(* LS Electric XG5000 project: test cps *)
(* PLC LSPLC *)
(* module base 0 slot 0: FEnet:XGL-EFMT(B) (Fast Ethernet 통신 모듈, 전기 Master) *)
VAR_GLOBAL
    T0 : TON;
    T1 : TON;
    T2 : TON;
    T3 : TON;
    T4 : TON;
    TP0 : TP;
    TP1 : TP;
    TP2 : TP;
    TP3 : TP;
END_VAR

(* Comments on direct variables
%MW0	1 comID
%MW1	2 comID
%MW2	3 comID
%MW3	4 comID
%MW4	5 comID
%MW5	6 comID
%MW6	7 comID
%MW7	8 comID
%MW8	1 Status
%MW9	2 Status
%MW10	3 Status
%MW11	4 Status
%MW12	5 Status
%MW13	6 Status
%MW14	7 Status
%MW15	8 Status
%MW16	1 ReadData
%MW17	2 ReadData
%MW18	3 ReadData
%MW19	4 ReadData
%MW20	5 ReadData
%MW21	6 ReadData
%MW22	7 ReadData
%MW23	8 ReadData
%MW101	1번무게합
%MW102	2번무게합
%MW103	3번무게합
%MW104	4번무게합
%MW201	리셋수(트레일러)
%MW202	리셋수(트레일러)
%MW203	리셋수(트레일러)
%MW204	리셋수(트레일러)
%QX0.0.0	Belt Conveyor 0
%QX0.0.1	Belt Conveyor 1
%QX0.0.2	Belt Conveyor 2
%QX0.0.3	box
%QX0.0.4	Belt Conveyor 4
%QX0.0.5	Belt Conveyor 5
%QX0.0.6	Belt Conveyor 6
%QX0.0.7	Belt Conveyor 7
%QX0.0.8	Belt Conveyor 8
%QX0.0.9	Belt Conveyor 9
%QX0.0.10	Belt Conveyor 10
%QX0.0.11	Belt Conveyor 11
%QX0.0.12	box
%QX0.0.13	Push 01
%QX0.0.14	Push 02
%QX0.0.15	Push 03
%QX0.0.16	Push 04
%QX0.0.17	0 Exexute
%QX0.0.18	1 Exexute
%QX0.0.19	2 Exexute
%QX0.0.20	3 Exexute
%QX0.0.21	4 Exexute
%QX0.0.22	5 Exexute
%QX0.0.23	6 Exexute
%QX0.0.24	7 Exexute
%QX0.0.25	8 Exexute
%QX0.0.26	9 Exexute
%IX0.0.0	Paused
%IX0.0.1	Reset
%IX0.0.2	Running
%IX0.0.3	write00
%IX0.0.4	write01
%IX0.0.5	1 Diffuse
%IX0.0.6	2 Diffuse
%IX0.0.7	3 Diffuse
%IX0.0.8	4 Diffuse
%IX0.0.9	5 Diffuse
%IX0.0.10	6 Diffuse
%IX0.0.11	7 Diffuse
%IX0.0.12	8 Diffuse
%IX0.0.13	1 Push front_lim
%IX0.0.14	2 Push front_lim
%IX0.0.15	3 Push front_lim
%IX0.0.16	4 Push front_lim
%WW0	0 command = write
%WW1	0 WriteData
%WW2	0 Memory Index
%WW3	9 command = write
%WW4	9 WriteData
%WW5	9 Memory Index
%WW6	1 command = Read
%WW7	1 Memory Index
%WW8	2 command = Read
%WW9	2 Memory Index
%WW10	3 command = Read
%WW11	3 Memory Index
%WW12	4 command = Read
%WW13	4 Memory Index
%WW14	5 command = Read
%WW15	5 Memory Index
%WW16	6 command = Read
%WW17	6 Memory Index
%WW18	7 command = Read
%WW19	7 Memory Index
%WW20	8 command = Read
%WW21	8 Memory Index
*)

PROGRAM NewProgram (* task: 스캔 프로그램 *)
VAR
    D0 : INT;
    D10 : INT;
    D100 : INT;
    D20 : INT;
    D200 : INT;
    sensor_0ff : TON;
    sensor_1ff : TON;
END_VAR
VAR_EXTERNAL
    T0 : TON;
    T1 : TON;
    T2 : TON;
    T3 : TON;
    T4 : TON;
    TP0 : TP;
    TP1 : TP;
    TP2 : TP;
    TP3 : TP;
END_VAR
VAR
    _t1 : BOOL;
    _t2 : BOOL;
    _t3 : BOOL;
    _t4 : BOOL;
    _t5 : BOOL;
    _t6 : BOOL;
    _t7 : BOOL;
    _t8 : BOOL;
    _t9 : BOOL;
    _e10 : R_TRIG;
    _t11 : BOOL;
    _e12 : R_TRIG;
    _t13 : BOOL;
    _e14 : R_TRIG;
    _t15 : BOOL;
    _e16 : R_TRIG;
END_VAR

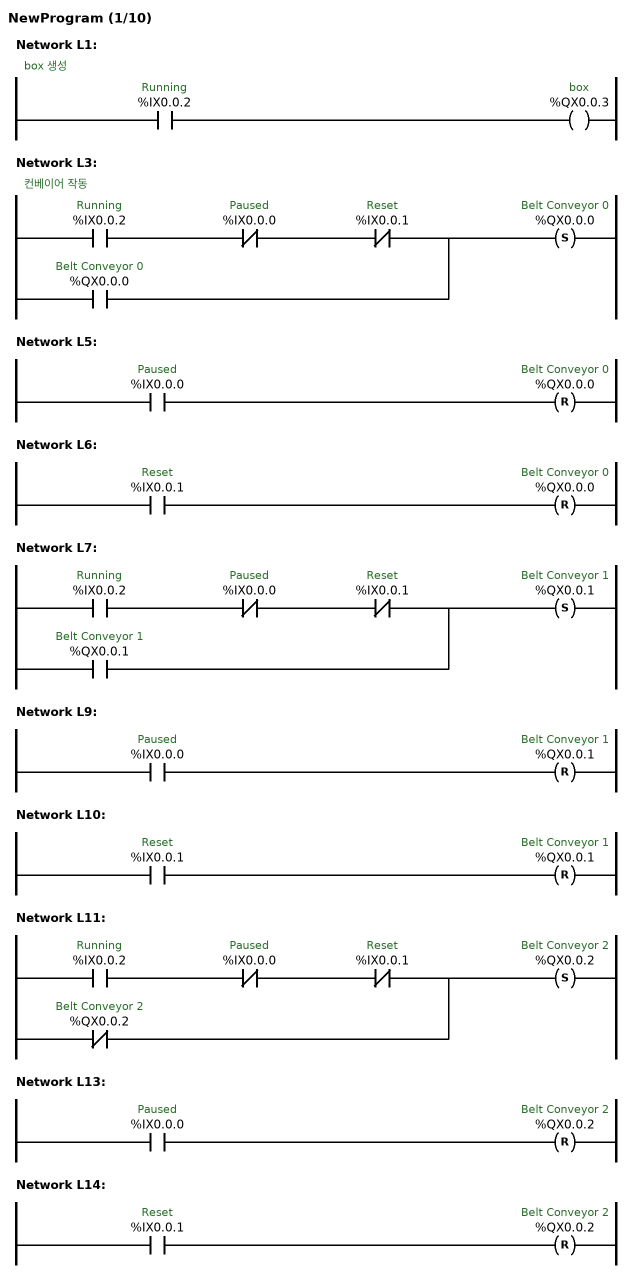
(* box 생성 *)
(* Rung L1 *)
%QX0.0.3 := %IX0.0.2;
(* 컨베이어 작동 *)
(* Rung L3 *)
IF (%IX0.0.2 AND NOT %IX0.0.0 AND NOT %IX0.0.1) OR %QX0.0.0 THEN %QX0.0.0 := TRUE; END_IF;
(* Rung L5 *)
IF %IX0.0.0 THEN %QX0.0.0 := FALSE; END_IF;
(* Rung L6 *)
IF %IX0.0.1 THEN %QX0.0.0 := FALSE; END_IF;
(* Rung L7 *)
IF (%IX0.0.2 AND NOT %IX0.0.0 AND NOT %IX0.0.1) OR %QX0.0.1 THEN %QX0.0.1 := TRUE; END_IF;
(* Rung L9 *)
IF %IX0.0.0 THEN %QX0.0.1 := FALSE; END_IF;
(* Rung L10 *)
IF %IX0.0.1 THEN %QX0.0.1 := FALSE; END_IF;
(* Rung L11 *)
IF (%IX0.0.2 AND NOT %IX0.0.0 AND NOT %IX0.0.1) OR NOT %QX0.0.2 THEN %QX0.0.2 := TRUE; END_IF;
(* Rung L13 *)
IF %IX0.0.0 THEN %QX0.0.2 := FALSE; END_IF;
(* Rung L14 *)
IF %IX0.0.1 THEN %QX0.0.2 := FALSE; END_IF;

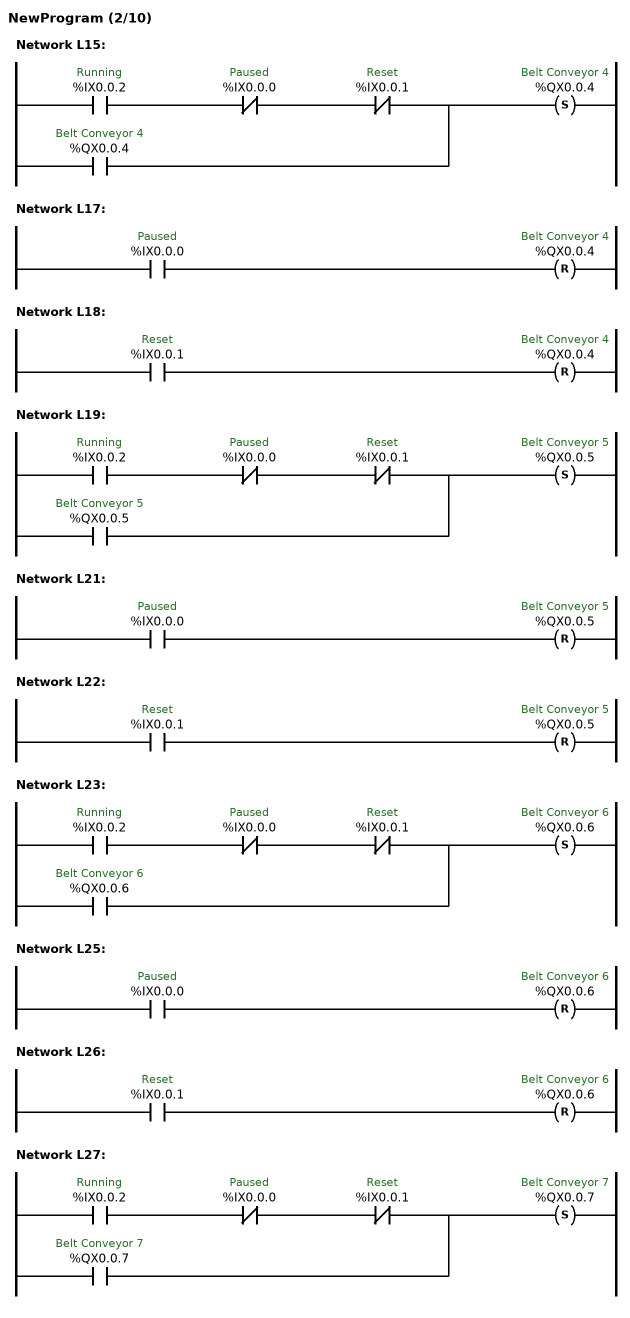
(* Rung L15 *)
IF (%IX0.0.2 AND NOT %IX0.0.0 AND NOT %IX0.0.1) OR %QX0.0.4 THEN %QX0.0.4 := TRUE; END_IF;
(* Rung L17 *)
IF %IX0.0.0 THEN %QX0.0.4 := FALSE; END_IF;
(* Rung L18 *)
IF %IX0.0.1 THEN %QX0.0.4 := FALSE; END_IF;
(* Rung L19 *)
IF (%IX0.0.2 AND NOT %IX0.0.0 AND NOT %IX0.0.1) OR %QX0.0.5 THEN %QX0.0.5 := TRUE; END_IF;
(* Rung L21 *)
IF %IX0.0.0 THEN %QX0.0.5 := FALSE; END_IF;
(* Rung L22 *)
IF %IX0.0.1 THEN %QX0.0.5 := FALSE; END_IF;
(* Rung L23 *)
IF (%IX0.0.2 AND NOT %IX0.0.0 AND NOT %IX0.0.1) OR %QX0.0.6 THEN %QX0.0.6 := TRUE; END_IF;
(* Rung L25 *)
IF %IX0.0.0 THEN %QX0.0.6 := FALSE; END_IF;
(* Rung L26 *)
IF %IX0.0.1 THEN %QX0.0.6 := FALSE; END_IF;
(* Rung L27 *)
IF (%IX0.0.2 AND NOT %IX0.0.0 AND NOT %IX0.0.1) OR %QX0.0.7 THEN %QX0.0.7 := TRUE; END_IF;

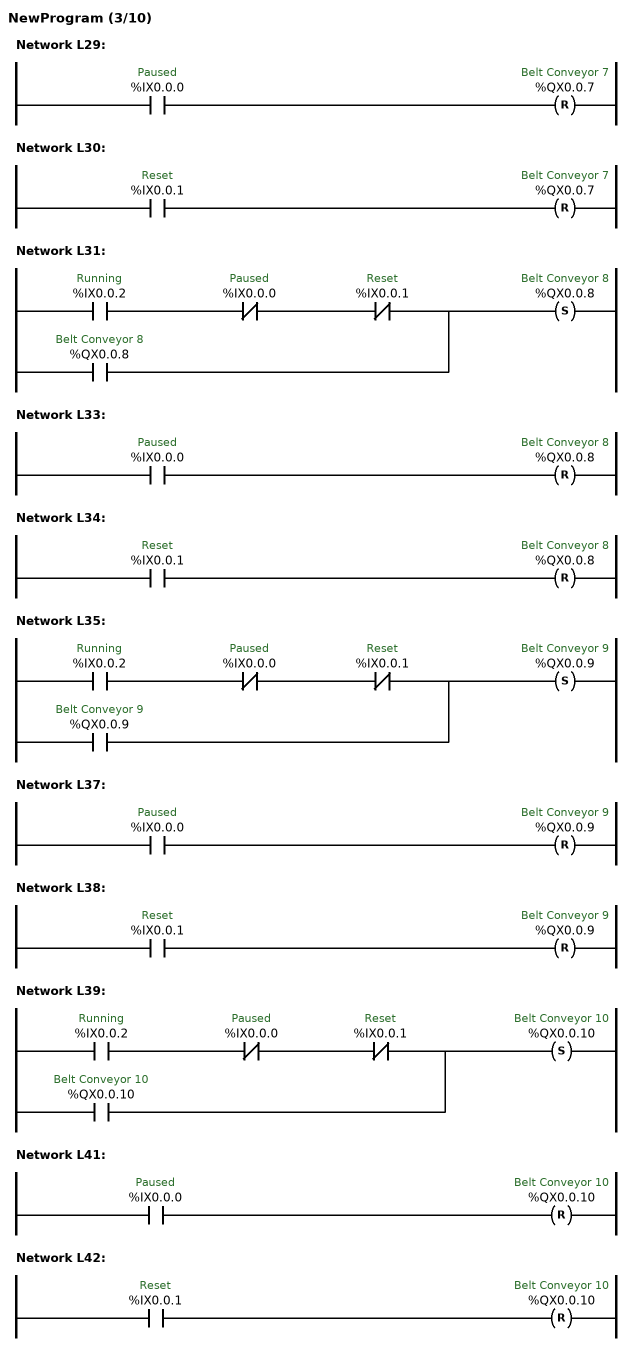
(* Rung L29 *)
IF %IX0.0.0 THEN %QX0.0.7 := FALSE; END_IF;
(* Rung L30 *)
IF %IX0.0.1 THEN %QX0.0.7 := FALSE; END_IF;
(* Rung L31 *)
IF (%IX0.0.2 AND NOT %IX0.0.0 AND NOT %IX0.0.1) OR %QX0.0.8 THEN %QX0.0.8 := TRUE; END_IF;
(* Rung L33 *)
IF %IX0.0.0 THEN %QX0.0.8 := FALSE; END_IF;
(* Rung L34 *)
IF %IX0.0.1 THEN %QX0.0.8 := FALSE; END_IF;
(* Rung L35 *)
IF (%IX0.0.2 AND NOT %IX0.0.0 AND NOT %IX0.0.1) OR %QX0.0.9 THEN %QX0.0.9 := TRUE; END_IF;
(* Rung L37 *)
IF %IX0.0.0 THEN %QX0.0.9 := FALSE; END_IF;
(* Rung L38 *)
IF %IX0.0.1 THEN %QX0.0.9 := FALSE; END_IF;
(* Rung L39 *)
IF (%IX0.0.2 AND NOT %IX0.0.0 AND NOT %IX0.0.1) OR %QX0.0.10 THEN %QX0.0.10 := TRUE; END_IF;
(* Rung L41 *)
IF %IX0.0.0 THEN %QX0.0.10 := FALSE; END_IF;
(* Rung L42 *)
IF %IX0.0.1 THEN %QX0.0.10 := FALSE; END_IF;

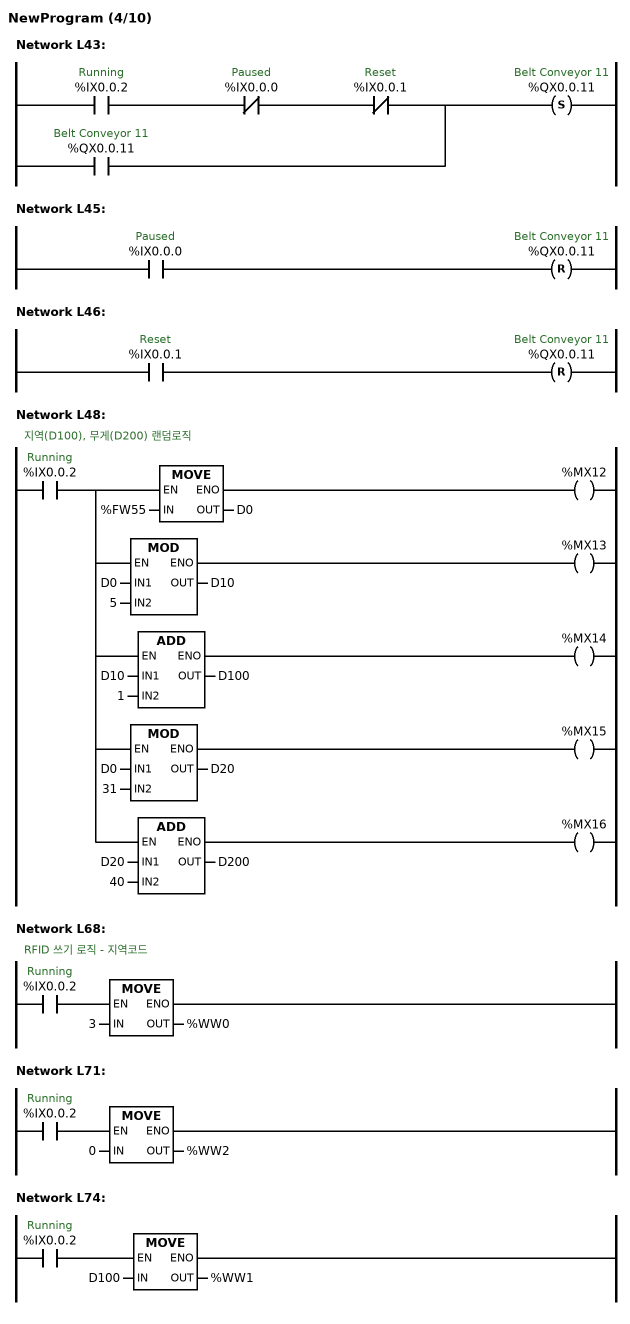
(* Rung L43 *)
IF (%IX0.0.2 AND NOT %IX0.0.0 AND NOT %IX0.0.1) OR %QX0.0.11 THEN %QX0.0.11 := TRUE; END_IF;
(* Rung L45 *)
IF %IX0.0.0 THEN %QX0.0.11 := FALSE; END_IF;
(* Rung L46 *)
IF %IX0.0.1 THEN %QX0.0.11 := FALSE; END_IF;
(* 지역(D100), 무게(D200) 랜덤로직 *)
(* Rung L48 *)
IF %IX0.0.2 THEN D0 := %FW55; END_IF;
%MX12 := %IX0.0.2;
IF %IX0.0.2 THEN D10 := D0 MOD 5; END_IF;
%MX13 := %IX0.0.2;
IF %IX0.0.2 THEN D100 := D10 + 1; END_IF;
%MX14 := %IX0.0.2;
IF %IX0.0.2 THEN D20 := D0 MOD 31; END_IF;
%MX15 := %IX0.0.2;
IF %IX0.0.2 THEN D200 := D20 + 40; END_IF;
%MX16 := %IX0.0.2;
(* RFID 쓰기 로직 - 지역코드 *)
(* Rung L68 *)
IF %IX0.0.2 THEN %WW0 := 3; END_IF;
(* Rung L71 *)
IF %IX0.0.2 THEN %WW2 := 0; END_IF;
(* Rung L74 *)
IF %IX0.0.2 THEN %WW1 := D100; END_IF;

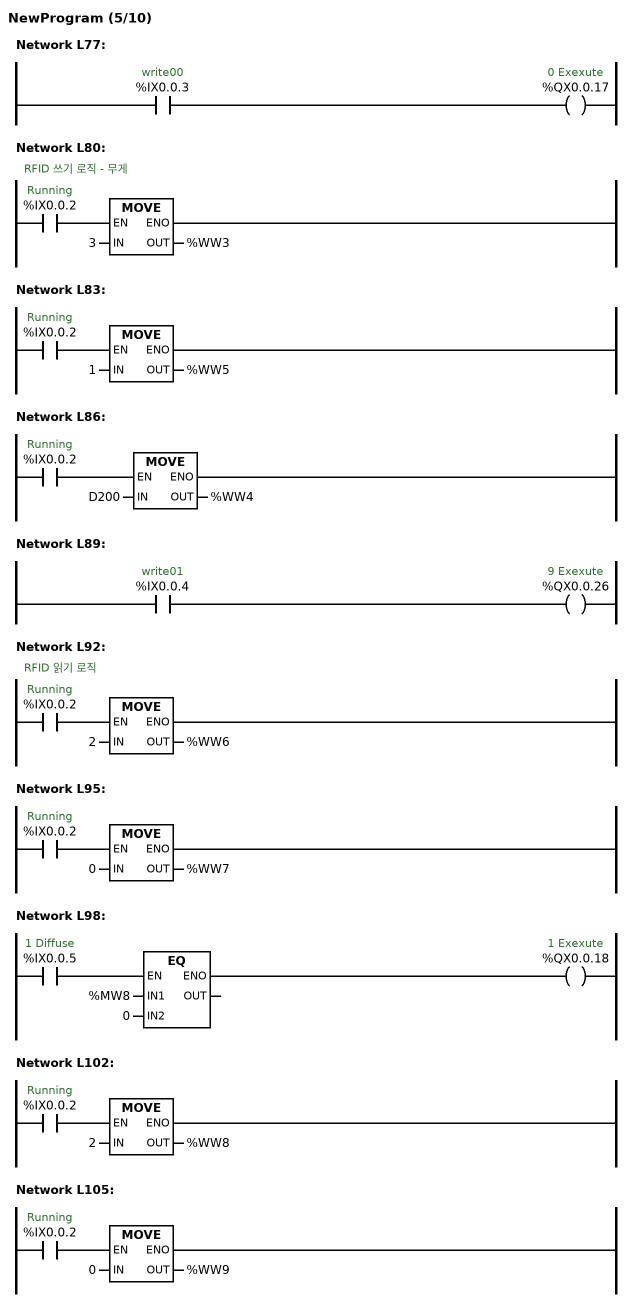
(* Rung L77 *)
%QX0.0.17 := %IX0.0.3;
(* RFID 쓰기 로직 - 무게 *)
(* Rung L80 *)
IF %IX0.0.2 THEN %WW3 := 3; END_IF;
(* Rung L83 *)
IF %IX0.0.2 THEN %WW5 := 1; END_IF;
(* Rung L86 *)
IF %IX0.0.2 THEN %WW4 := D200; END_IF;
(* Rung L89 *)
%QX0.0.26 := %IX0.0.4;
(* RFID 읽기 로직 *)
(* Rung L92 *)
IF %IX0.0.2 THEN %WW6 := 2; END_IF;
(* Rung L95 *)
IF %IX0.0.2 THEN %WW7 := 0; END_IF;
(* Rung L98 *)
IF %IX0.0.5 THEN _t1 := %MW8 = 0; END_IF;
%QX0.0.18 := %IX0.0.5;
(* Rung L102 *)
IF %IX0.0.2 THEN %WW8 := 2; END_IF;
(* Rung L105 *)
IF %IX0.0.2 THEN %WW9 := 0; END_IF;

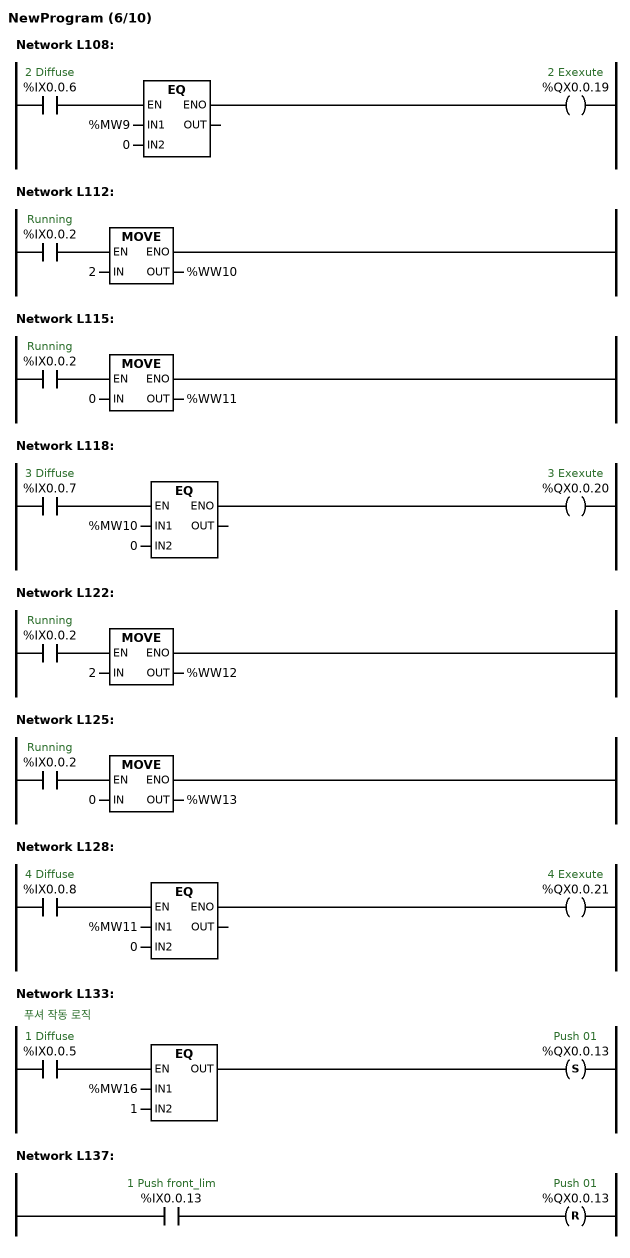
(* Rung L108 *)
IF %IX0.0.6 THEN _t2 := %MW9 = 0; END_IF;
%QX0.0.19 := %IX0.0.6;
(* Rung L112 *)
IF %IX0.0.2 THEN %WW10 := 2; END_IF;
(* Rung L115 *)
IF %IX0.0.2 THEN %WW11 := 0; END_IF;
(* Rung L118 *)
IF %IX0.0.7 THEN _t3 := %MW10 = 0; END_IF;
%QX0.0.20 := %IX0.0.7;
(* Rung L122 *)
IF %IX0.0.2 THEN %WW12 := 2; END_IF;
(* Rung L125 *)
IF %IX0.0.2 THEN %WW13 := 0; END_IF;
(* Rung L128 *)
IF %IX0.0.8 THEN _t4 := %MW11 = 0; END_IF;
%QX0.0.21 := %IX0.0.8;
(* 푸셔 작동 로직 *)
(* Rung L133 *)
IF %IX0.0.5 THEN _t5 := %MW16 = 1; END_IF;
IF _t5 THEN %QX0.0.13 := TRUE; END_IF;
(* Rung L137 *)
IF %IX0.0.13 THEN %QX0.0.13 := FALSE; END_IF;

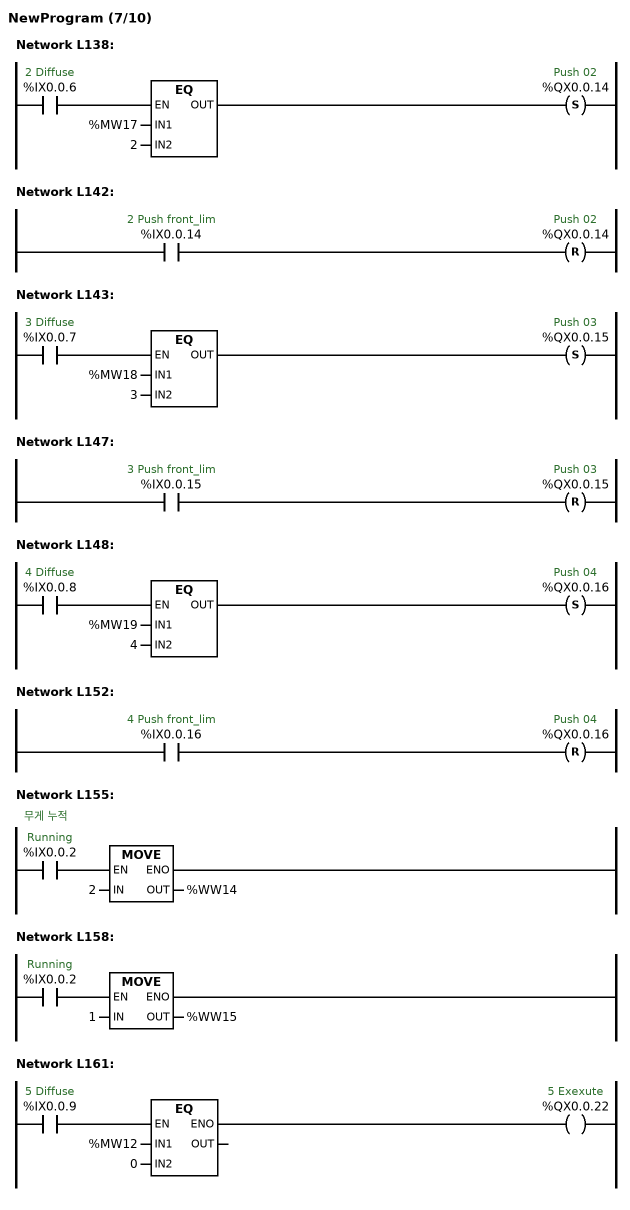
(* Rung L138 *)
IF %IX0.0.6 THEN _t6 := %MW17 = 2; END_IF;
IF _t6 THEN %QX0.0.14 := TRUE; END_IF;
(* Rung L142 *)
IF %IX0.0.14 THEN %QX0.0.14 := FALSE; END_IF;
(* Rung L143 *)
IF %IX0.0.7 THEN _t7 := %MW18 = 3; END_IF;
IF _t7 THEN %QX0.0.15 := TRUE; END_IF;
(* Rung L147 *)
IF %IX0.0.15 THEN %QX0.0.15 := FALSE; END_IF;
(* Rung L148 *)
IF %IX0.0.8 THEN _t8 := %MW19 = 4; END_IF;
IF _t8 THEN %QX0.0.16 := TRUE; END_IF;
(* Rung L152 *)
IF %IX0.0.16 THEN %QX0.0.16 := FALSE; END_IF;
(* 무게 누적 *)
(* Rung L155 *)
IF %IX0.0.2 THEN %WW14 := 2; END_IF;
(* Rung L158 *)
IF %IX0.0.2 THEN %WW15 := 1; END_IF;
(* Rung L161 *)
IF %IX0.0.9 THEN _t9 := %MW12 = 0; END_IF;
%QX0.0.22 := %IX0.0.9;

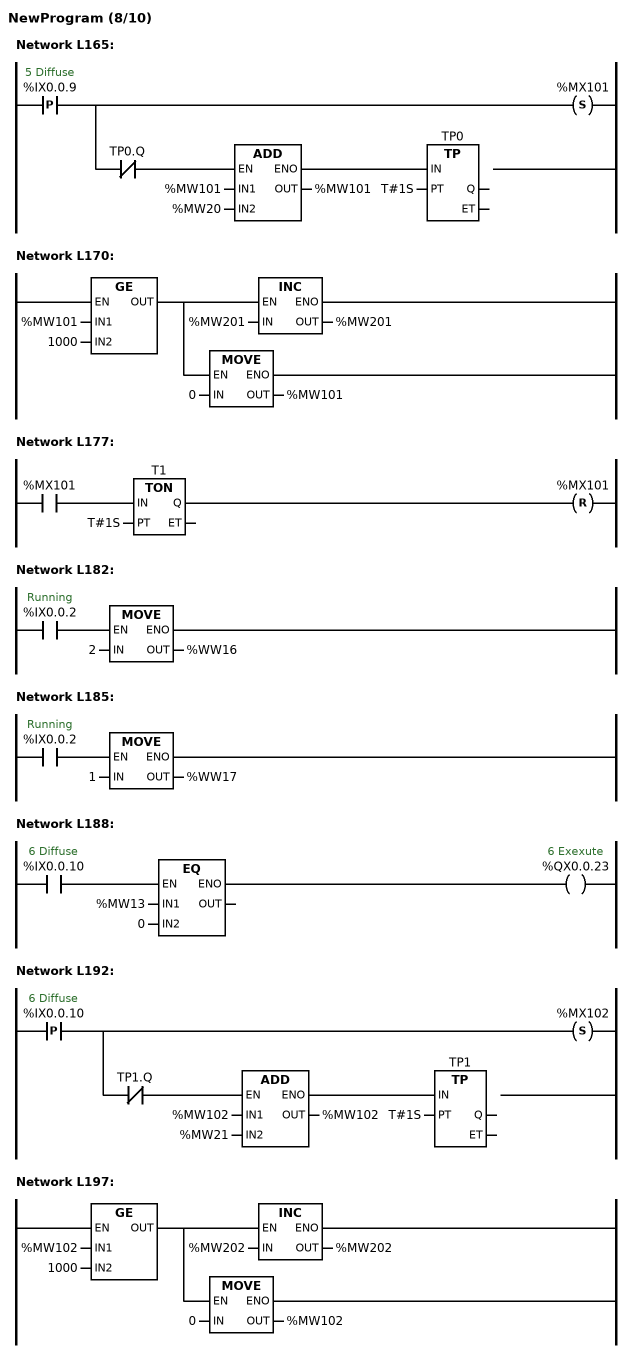
(* Rung L165 *)
_e10(CLK := %IX0.0.9);
IF _e10.Q THEN %MX101 := TRUE; END_IF;
IF _e10.Q AND NOT TP0.Q THEN %MW101 := %MW101 + %MW20; END_IF;
TP0(IN := _e10.Q AND NOT TP0.Q, PT := T#1S);
(* Rung L170 *)
IF %MW101 >= 1000 THEN
    %MW201 := INC(%MW201);
    %MW101 := 0;
END_IF;
(* Rung L177 *)
T1(IN := %MX101, PT := T#1S);
IF T1.Q THEN %MX101 := FALSE; END_IF;
(* Rung L182 *)
IF %IX0.0.2 THEN %WW16 := 2; END_IF;
(* Rung L185 *)
IF %IX0.0.2 THEN %WW17 := 1; END_IF;
(* Rung L188 *)
IF %IX0.0.10 THEN _t11 := %MW13 = 0; END_IF;
%QX0.0.23 := %IX0.0.10;
(* Rung L192 *)
_e12(CLK := %IX0.0.10);
IF _e12.Q THEN %MX102 := TRUE; END_IF;
IF _e12.Q AND NOT TP1.Q THEN %MW102 := %MW102 + %MW21; END_IF;
TP1(IN := _e12.Q AND NOT TP1.Q, PT := T#1S);
(* Rung L197 *)
IF %MW102 >= 1000 THEN
    %MW202 := INC(%MW202);
    %MW102 := 0;
END_IF;

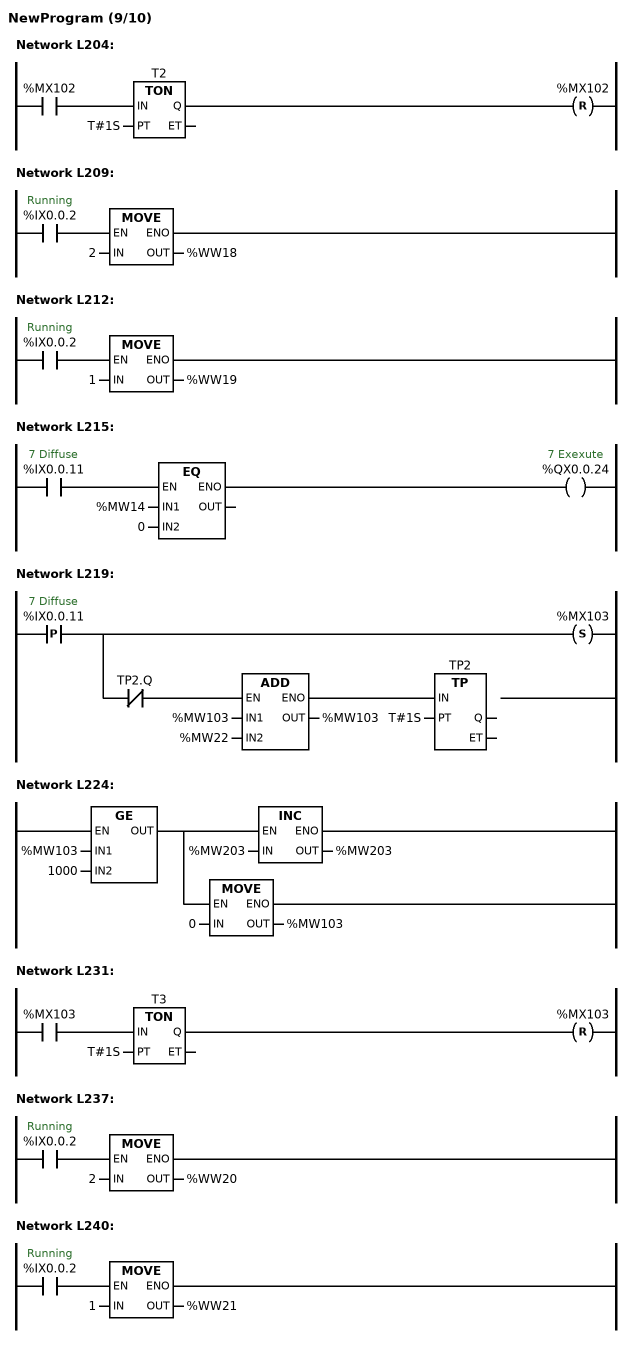
(* Rung L204 *)
T2(IN := %MX102, PT := T#1S);
IF T2.Q THEN %MX102 := FALSE; END_IF;
(* Rung L209 *)
IF %IX0.0.2 THEN %WW18 := 2; END_IF;
(* Rung L212 *)
IF %IX0.0.2 THEN %WW19 := 1; END_IF;
(* Rung L215 *)
IF %IX0.0.11 THEN _t13 := %MW14 = 0; END_IF;
%QX0.0.24 := %IX0.0.11;
(* Rung L219 *)
_e14(CLK := %IX0.0.11);
IF _e14.Q THEN %MX103 := TRUE; END_IF;
IF _e14.Q AND NOT TP2.Q THEN %MW103 := %MW103 + %MW22; END_IF;
TP2(IN := _e14.Q AND NOT TP2.Q, PT := T#1S);
(* Rung L224 *)
IF %MW103 >= 1000 THEN
    %MW203 := INC(%MW203);
    %MW103 := 0;
END_IF;
(* Rung L231 *)
T3(IN := %MX103, PT := T#1S);
IF T3.Q THEN %MX103 := FALSE; END_IF;
(* Rung L237 *)
IF %IX0.0.2 THEN %WW20 := 2; END_IF;
(* Rung L240 *)
IF %IX0.0.2 THEN %WW21 := 1; END_IF;

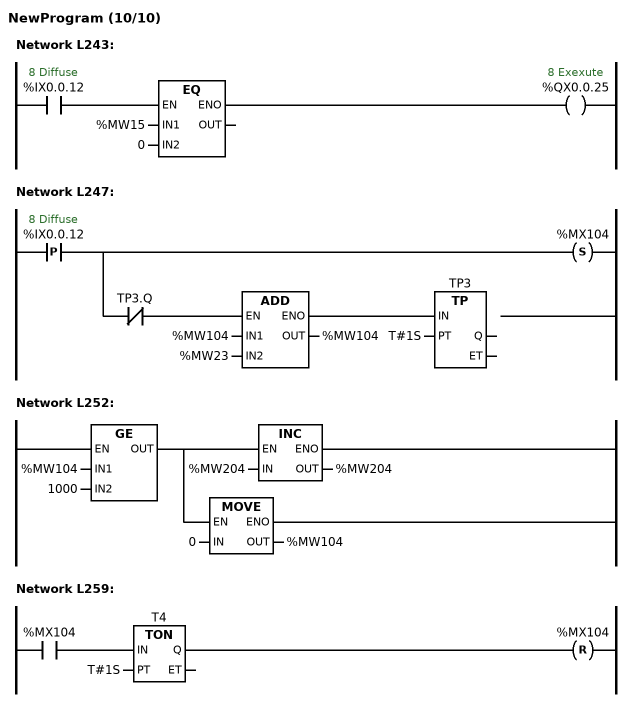
(* Rung L243 *)
IF %IX0.0.12 THEN _t15 := %MW15 = 0; END_IF;
%QX0.0.25 := %IX0.0.12;
(* Rung L247 *)
_e16(CLK := %IX0.0.12);
IF _e16.Q THEN %MX104 := TRUE; END_IF;
IF _e16.Q AND NOT TP3.Q THEN %MW104 := %MW104 + %MW23; END_IF;
TP3(IN := _e16.Q AND NOT TP3.Q, PT := T#1S);
(* Rung L252 *)
IF %MW104 >= 1000 THEN
    %MW204 := INC(%MW204);
    %MW104 := 0;
END_IF;
(* Rung L259 *)
T4(IN := %MX104, PT := T#1S);
IF T4.Q THEN %MX104 := FALSE; END_IF;
END_PROGRAM